(* IEC 61131-3 sources: programs/VI-54/VI-54_20171205/VI-54_20171205/Stations/Screen/LseClass170718/Class/FileTransfer, 1 file *)

(* ---- FileTransfer.st ---- *)
(*!
<Class
	Name               = "FileTransfer"
	Revision           = "1.2"
	RealtimeTask       = "false"
	CyclicTask         = "false"
	BackgroundTask     = "false"
	Sigmatek           = "false"
	OSInterface        = "false"
	HighPriority       = "false"
	Automatic          = "false"
	UpdateMode         = "Prescan"
	SharedCommandTable = "true"
	Objectsize         = "(1050,420)"
	Comment            = "Die Klasse dient dem Austausch von&#13;&#10;Files zwischen zwei CPUs bzw.Terminals.&#13;&#10;Kann verwendet werden um Files&#13;&#10;von einer 2ten CPU zu holen.&#13;&#10;Die Klasse alleine ist nicht funktionsfähig. Sie benötigt&#13;&#10;die Klasse DataMng um korrekt zu funktionieren.">
	<Channels>
		<Server Name="ClassSvr" Visualized="false" Initialize="false" WriteProtected="true" Retentive="false" Comment="Objekt-Server der Klasse. Der Client cFileTransfer der Klasse&#13;&#10;FolderTransfer muss hierher verbunden werden wenn man diese nutzt.&#13;&#10;Ansonsten kann man den Status der letzten Operation mit der Methode&#13;&#10;GetStateOfProcess abgefragt werden."/>
		<Server Name="sDestinationID" Visualized="false" Initialize="true" WriteProtected="true" Retentive="false" Comment="Destination communication id number."/>
		<Server Name="sErrorNr" Visualized="true" Initialize="false" WriteProtected="true" Retentive="false" Comment="Interne Fehlernummer."/>
		<Server Name="sMyID" Visualized="false" Initialize="true" WriteProtected="true" Retentive="false" Comment="Source communication id number."/>
		<Server Name="sState" Class="FileTransferHandle" Visualized="true" Initialize="false" WriteProtected="true" Retentive="false" Comment="Status des letzten Kommandos ."/>
		<Server Name="sSubState" Visualized="true" Initialize="false" WriteProtected="true" Retentive="false" Comment="Genauere Aufschlüsselung des aktuell durchlaufenen Schritts"/>
		<Client Name="cDataManager" Required="true" Internal="false" Comment="Connection to communication data manager."/>
		<Client Name="cPrio" Required="true" Internal="false" Comment="Communication priority number."/>
		<Client Name="FileTransferHandle" Required="true" Internal="true"/>
		<Client Name="RecvData" Required="true" Internal="true"/>
		<Client Name="SendData" Required="true" Internal="true"/>
	</Channels>
	<Dependencies>
		<Files>
			<File Path=".\Class\FileTransfer\FileTransfer.pdf"/>
			<File Path=".\Class\FileTransfer\Diagnostic_Def.h" Include="true"/>
		</Files>
	</Dependencies>
	<RevDoku>
		<Owner Company="Sigmatek" Author="hötant"/>
		<Dokumentation Revision="1.2" Date="2015-10-27" Author="hötant" Company="Sigmatek" Description="added documentation file"/>
		<Dokumentation Revision="1.1" Date="2015-10-21" Author="hötant" Company="Sigmatek" Description="added error handling and some improvements"/>
		<Dokumentation Revision="1.0" Date="2015-10-15" Author="hötant" Company="Sigmatek" Description="creation of class"/>
	</RevDoku>
	<Network Name="FileTransfer">
		<!-- List of Components in this network -->
		<Components>
			<Object
				Name           = "FileTransferHandle"
				Class          = "FileTransferHandle"
				Position       = "(1080,360)"
				Visualized     = "false"
				BackgroundTime = "100 ms">
				<Channels>
					<Server Name="sCallbackError"/>
					<Server Name="sCallbackOK"/>
					<Server Name="sErrorNr"/>
					<Server Name="sState"/>
					<Server Name="sSubState"/>
					<Client Name="cFileSys"/>
					<Client Name="cGrafix"/>
					<Client Name="cSigCLib"/>
					<Client Name="cToCom"/>
				</Channels>
			</Object>
			<Object
				Name       = "RecvData"
				Class      = "FileTransfer_RecvData"
				Position   = "(2010,120)"
				Visualized = "false">
				<Channels>
					<Server Name="ClassSvr"/>
					<Server Name="sMyID"/>
					<Server Name="sRecvCnt"/>
					<Client Name="cDataMng"/>
					<Client Name="cFileTransfer"/>
				</Channels>
			</Object>
			<Object
				Name       = "SendData"
				Class      = "Comm_SendData"
				Position   = "(360,360)"
				Visualized = "false">
				<Channels>
					<Server Name="ClassSvr"/>
					<Server Name="sDestinationId"/>
					<Server Name="sMyId"/>
					<Server Name="sSendCnt"/>
					<Server Name="sSendErr"/>
					<Client Name="cDataMng"/>
					<Client Name="cPrio"/>
					<Client Name="cSendErr"/>
					<Client Name="cSendOk"/>
				</Channels>
			</Object>
		</Components>
		<Comments>
		</Comments>
		<!-- List of Connections in this network -->
		<Connections>
			<Connection Source="this.RecvData" Destination="RecvData.ClassSvr"/>
			<Connection Source="this.FileTransferHandle" Destination="FileTransferHandle.sState"/>
			<Connection Source="this.SendData" Destination="SendData.ClassSvr"/>
			<Connection Source="RecvData.cFileTransfer" Destination="FileTransferHandle.sState" Vertices="(2010,270),(1920,270),(1920,450),(1726,450),"/>
			<Connection Source="FileTransferHandle.cToCom" Destination="SendData.ClassSvr" Vertices="(1080,450),(976,450),"/>
			<Connection Source="SendData.cDataMng" Destination="this.cDataManager" Vertices="(360,450),(270,450),(270,210),(38,210),"/>
			<Connection Source="RecvData.cDataMng" Destination="this.cDataManager" Vertices="(2010,210),(38,210),"/>
			<Connection Source="SendData.cPrio" Destination="this.cPrio" Vertices="(360,510),(180,510),(180,270),(38,270),"/>
			<Connection Source="SendData.cSendOk" Destination="FileTransferHandle.sCallbackOK" Vertices="(360,570),(180,570),(180,870),(1920,870),(1920,630),(1726,630),"/>
			<Connection Source="SendData.cSendErr" Destination="FileTransferHandle.sCallbackError" Vertices="(360,630),(270,630),(270,840),(1830,840),(1830,690),(1726,690),"/>
			<Connection Source="this.sState" Destination="FileTransferHandle.sState" Vertices="(2646,390),(2460,390),(2460,450),(1726,450),"/>
			<Connection Source="this.sSubState" Destination="FileTransferHandle.sSubState" Vertices="(2646,450),(2520,450),(2520,510),(1726,510),"/>
			<Connection Source="this.sErrorNr" Destination="FileTransferHandle.sErrorNr" Vertices="(2646,510),(2580,510),(2580,570),(1726,570),"/>
		</Connections>
		<!-- Headerfiles -->
		<Options>
		</Options>
	</Network>
</Class>
*)
FileTransfer : CLASS
  //Servers:
	ClassSvr 	: SvrChCmd_DINT;
	sMyID 	: SvrCh_DINT;
	sDestinationID 	: SvrCh_DINT;
	sState 	: SvrChCmd__FT_State_PTofCls_FileTransferHandle;
	sSubState 	: SvrCh__FT_SubState_PTofCls_FileTransferHandle;
	sErrorNr 	: SvrCh_DINT;
  //Clients:
	FileTransferHandle 	: CltChCmd_FileTransferHandle;
	cDataManager 	: CltChCmd_DataManager;
	cPrio 	: CltCh_DINT;
	SendData 	: CltChCmd_Comm_SendData;
	RecvData 	: CltChCmd_FileTransfer_RecvData;
  //Variables:
  //Functions:
				//! <Function Comment="Nicht für den Benutzer.( Initialisierung )" Name="Init"/>
	FUNCTION VIRTUAL GLOBAL Init;
				//! <Function Comment="Wird verwendet, um ein File von der Gegenstelle zu holen." Name="GetFile"/>
	FUNCTION GLOBAL GetFile
		VAR_INPUT
			pSourceDP 	: ^CHAR;			//! <Variable Comment="Laufwerk und Ordner des zu holenden Files ( z.B.: &quot;C:\Test\Hallo\&quot; )" Name="GetFile.pSourceDP"/>
			pSourceNE 	: ^CHAR;			//! <Variable Comment="Name und Endung des Files ( z.B.: &quot;logfile.dat&quot; )" Name="GetFile.pSourceNE"/>
			pDestinationDP 	: ^CHAR;			//! <Variable Comment="Laufwerk und Ordnername , wohin das File kopiert werden soll.&#13;&#10;( z.B.: &quot;E:\Export\&quot; ) Der Ordner muss bereits existieren." Name="GetFile.pDestinationDP"/>
		END_VAR
		VAR_OUTPUT
			retcode 	: DINT;			//! <Variable Comment="0 .. Es läuft bereits eine andere Aktion&#13;&#10;1 .. Transfer wurde erfolgreich gestartet.&#13;&#10;-1 .. Einer der übergebenen Pointer ist NULL&#13;&#10;-2 .. Befehl konnte der Kommunikation nicht weitergegeben werden." Name="GetFile.retcode"/>
		END_VAR;
				//! <Function Comment="Wird verwendet, um den Status der letzten Aktion zu überprüfen." Name="GetStateOfProcess"/>
	FUNCTION GLOBAL GetStateOfProcess
		VAR_OUTPUT
			retcode 	: FileTransferHandle::_FT_State;			//! <Variable Comment="FT_NoAction .. aktuelle keine Aktive Aktion&#13;&#10;FT_OperationReady .. Aktion wurde ohne Fehler durchgeführt.&#13;&#10;FT_Error .. Es ist ein Fehler aufgetreten.&#13;&#10;&#13;&#10;Der Server sSubState gibt genauere Auskünfte über Fehler oder&#13;&#10;aktuelle Statusinformationen." Name="GetStateOfProcess.retcode"/>
		END_VAR;
  //Tables:
	FUNCTION @STD
		VAR_OUTPUT
			ret_code	: CONFSTATES;
		END_VAR;
	FUNCTION GLOBAL TAB @CT_;
END_CLASS;

#pragma using Comm_SendData
#pragma using FileTransfer_RecvData
#pragma using FileTransferHandle
#pragma usingLtd DataManager

FUNCTION VIRTUAL GLOBAL FileTransfer::Init

  // Initwerte übernehmen
  SendData.sMyId := sMyID;
  SendData.sDestinationId := sDestinationID;
  RecvData.sMyID := sMyID;

END_FUNCTION

FUNCTION GLOBAL FileTransfer::GetFile
	VAR_INPUT
		pSourceDP 	: ^CHAR;
		pSourceNE 	: ^CHAR;
    pDestinationDP 	: ^CHAR;
	END_VAR
	VAR_OUTPUT
		retcode 	: DINT;
	END_VAR

  // Funktion weiterleiten.
  retcode := FileTransferHandle.GetFile(pSourceDP, pSourceNE,pDestinationDP);

END_FUNCTION

FUNCTION GLOBAL FileTransfer::GetStateOfProcess
	VAR_OUTPUT
		retcode 	: FileTransferHandle::_FT_State;
	END_VAR

  // aktuellen status zurückgeben.
  retcode := FileTransferHandle.sState;

END_FUNCTION
